// TIA Portal V19 export
FUNCTION "Pb_CIP_With_Lye_Only" : Void   // FC61, STL
TITLE = Pb - CIP WITH LYE ONLY
{ S7_Optimized_Access := 'TRUE' }
NAME : PBLYECIP
VERSION : 0.0
// Comment
// stored: AutoNumber false
   VAR_TEMP
      alarmbit : Int;
   END_VAR
BEGIN

NETWORK
TITLE = Pb - CIP WITH LYE ONLY
      AN    "LEDAssignment".K4_BUTTON;  // "PbK4CipLye"
      BEC;
      R     "LEDAssignment".K4_BUTTON;  // "PbK4CipLye"
      A     "S0 FILLER";
      S     "ProcessAndPbAlarms"."A"[6];  //A06_CipFillerStarted//  _CIP_FILLER_STARTED
      L     6;
      JC    Alrm;

//      BEC
      A     "S0 CHAIN WASH";
      S     "ProcessAndPbAlarms"."A"[7];  //A07_CipUnitOccupied// cip unit occupied
      L     7;
      JC    Alrm;

//      BEC
      A     "TANK AUTO";
      JC    M001;
      AN    "PA0572_Air";
      S     "ProcessAndPbAlarms"."A"[3];  //A03_NoInstrumentAir// no intrument air
      L     3;
      JC    Alrm;

//      BEC
      AN    "PA0561_Steam";
      S     "ProcessAndPbAlarms"."A"[4];  //A04_NoSteam// no steam
      L     4;
      JC    Alrm;

//      BEC
      A     "DUMMY UPD.DRAIN TANK";
      S     "ProcessAndPbAlarms"."A"[5];  //A05_DrainIsActive// drain is active
      L     5;
      JC    Alrm;

//      BEC
      A(;
      AN    "GS22_61";
      A     "GS22_62";
      AN    "GS22_63";
      A     "GS22_68";
      O;
      A     "GS22_61";
      AN    "GS22_62";
      A     "GS22_63";
      AN    "GS22_68";
      );
      NOT;
      S     "ProcessAndPbAlarms"."A"[18];  //A18_SwingbendOutOfPosn// swingbend out of position
      L     6;
      JC    Alrm;

//      BEC
      S     "S0 CIP TANK";
      S     "LEDAssignment".K4_FLASH;  //"FLASH_K4_CIP_LYE"
      S     "LEDAssignment".K4_LIGHT;  //"LIGHT_K4_CIP_LYE"
      BEU;
M001: AN    "LEDAssignment".K4_FLASH;  //"FLASH_K4_CIP_LYE"
      S     "ProcessAndPbAlarms"."A"[8];  //A08_NotReadyForCip// not ready for cip
      L     8;
      JC    Alrm;

//      BEC
      S     "S0 CIP TANK";
      S     "LEDAssignment".K4_FLASH;  //"FLASH_K4_CIP_LYE"
      S     "LEDAssignment".K4_LIGHT;  //"LIGHT_K4_CIP_LYE"
      R     "LEDAssignment".K5_FLASH;  //"FLASH_K5_CIP_LYE_ACID"
      R     "LEDAssignment".K5_LIGHT;  //"LIGHT_K5_CIP_LYE_ACID"
      R     "S0 STOP PRODUCTION TANK";  // Rettet 21-05-96
      BEU;

NETWORK
TITLE = Blockings alarm text
// Blockings alarm
Alrm: NOP   1;
      T     #alarmbit;
      CALL  "Set_Pop_Up_Blocking"
      ( alarmTextNum := #alarmbit
      );  // start blockings text

END_FUNCTION
